// TIA Portal V16 export
// export: Created 2021-11-12T13:32:31.7441446Z, ExportSetting WithDefaults, DisplayName Totally Integrated Automation Portal, DisplayVersion V16 Update 3, DisplayName TIA Portal Version Control Interface, DisplayVersion V16 Update 2, DisplayName TIA Portal Openness, DisplayVersion V16 Update 3, DisplayName SINAMICS Startdrive Advanced, DisplayVersion V16 Update 5, DisplayName SINAMICS Startdrive G130, G150, S120, S150, SINAMICS MV, S210, DisplayVersion V16 Update 5, DisplayName SINAMICS Startdrive G110M, G120, G120C, G120D, G120P, G115D, DisplayVersion V16 Update 5, DisplayName STEP 7 Professional, DisplayVersion V16 Update 3, DisplayName STEP 7 Safety, DisplayVersion V16, DisplayName WinCC UA Professional, DisplayVersion V16 Update 3
FUNCTION_BLOCK "IM_100+UH13-KF10"   // FB62, LAD
TITLE = Inputs reading
{ S7_Optimized_Access := 'TRUE' }
VERSION : 0.1
// MICE Wood interface block
// stored: AutoNumber true, IsIECCheckEnabled false, IsRetainMemResEnabled false, MemoryReserve 100, SetENOAutomatically false, UDAEnableTagReadback false
   VAR
      KF11_Ix0 { S7_SetPoint := 'True'} : "STD_CH_DI";
      KF11_Ix1 { S7_SetPoint := 'True'} : "STD_CH_DI";
      KF11_Ix2 { S7_SetPoint := 'True'} : "STD_CH_DI";
      KF11_Ix3 { S7_SetPoint := 'True'} : "STD_CH_DI";
      KF11_Ix4 { S7_SetPoint := 'True'} : "STD_CH_DI";
      KF11_Ix5 { S7_SetPoint := 'True'} : "STD_CH_DI";
      KF11_Ix6 { S7_SetPoint := 'True'} : "STD_CH_DI";
      KF11_Ix7 { S7_SetPoint := 'True'} : "STD_CH_DI";
      KF11_Ix8 { S7_SetPoint := 'True'} : "STD_CH_DI";
      KF11_Ix9 { S7_SetPoint := 'True'} : "STD_CH_DI";
      KF11_Ix10 { S7_SetPoint := 'True'} : "STD_CH_DI";
      KF11_Ix11 { S7_SetPoint := 'True'} : "STD_CH_DI";
      KF11_Ix12 { S7_SetPoint := 'True'} : "STD_CH_DI";
      KF11_Ix13 { S7_SetPoint := 'True'} : "STD_CH_DI";
      KF11_Ix14 { S7_SetPoint := 'True'} : "STD_CH_DI";
      KF11_Ix15 { S7_SetPoint := 'True'} : "STD_CH_DI";
      KF12_Ix0 { S7_SetPoint := 'True'} : "STD_CH_DI";
      KF12_Ix1 { S7_SetPoint := 'True'} : "STD_CH_DI";
      KF12_Ix2 { S7_SetPoint := 'True'} : "STD_CH_DI";
      KF12_Ix3 { S7_SetPoint := 'True'} : "STD_CH_DI";
      KF12_Ix4 { S7_SetPoint := 'True'} : "STD_CH_DI";
      KF12_Ix5 { S7_SetPoint := 'True'} : "STD_CH_DI";
      KF12_Ix6 { S7_SetPoint := 'True'} : "STD_CH_DI";
      KF12_Ix7 { S7_SetPoint := 'True'} : "STD_CH_DI";
      KF12_Ix8 { S7_SetPoint := 'True'} : "STD_CH_DI";
      KF12_Ix9 { S7_SetPoint := 'True'} : "STD_CH_DI";
      KF12_Ix10 { S7_SetPoint := 'True'} : "STD_CH_DI";
      KF12_Ix11 { S7_SetPoint := 'True'} : "STD_CH_DI";
      KF12_Ix12 { S7_SetPoint := 'True'} : "STD_CH_DI";
      KF12_Ix13 { S7_SetPoint := 'True'} : "STD_CH_DI";
      KF12_Ix14 { S7_SetPoint := 'True'} : "STD_CH_DI";
      KF12_Ix15 { S7_SetPoint := 'True'} : "STD_CH_DI";
   END_VAR
   VAR_TEMP   // added for the SCL form of the ladder/FBD networks
      _w1 : Bool;
      _w2 : Bool;
      _w3 : Bool;
      _w4 : Bool;
      _w5 : Bool;
      _w6 : Bool;
      _w7 : Bool;
   END_VAR
BEGIN

REGION Network 1: Module position -KF11
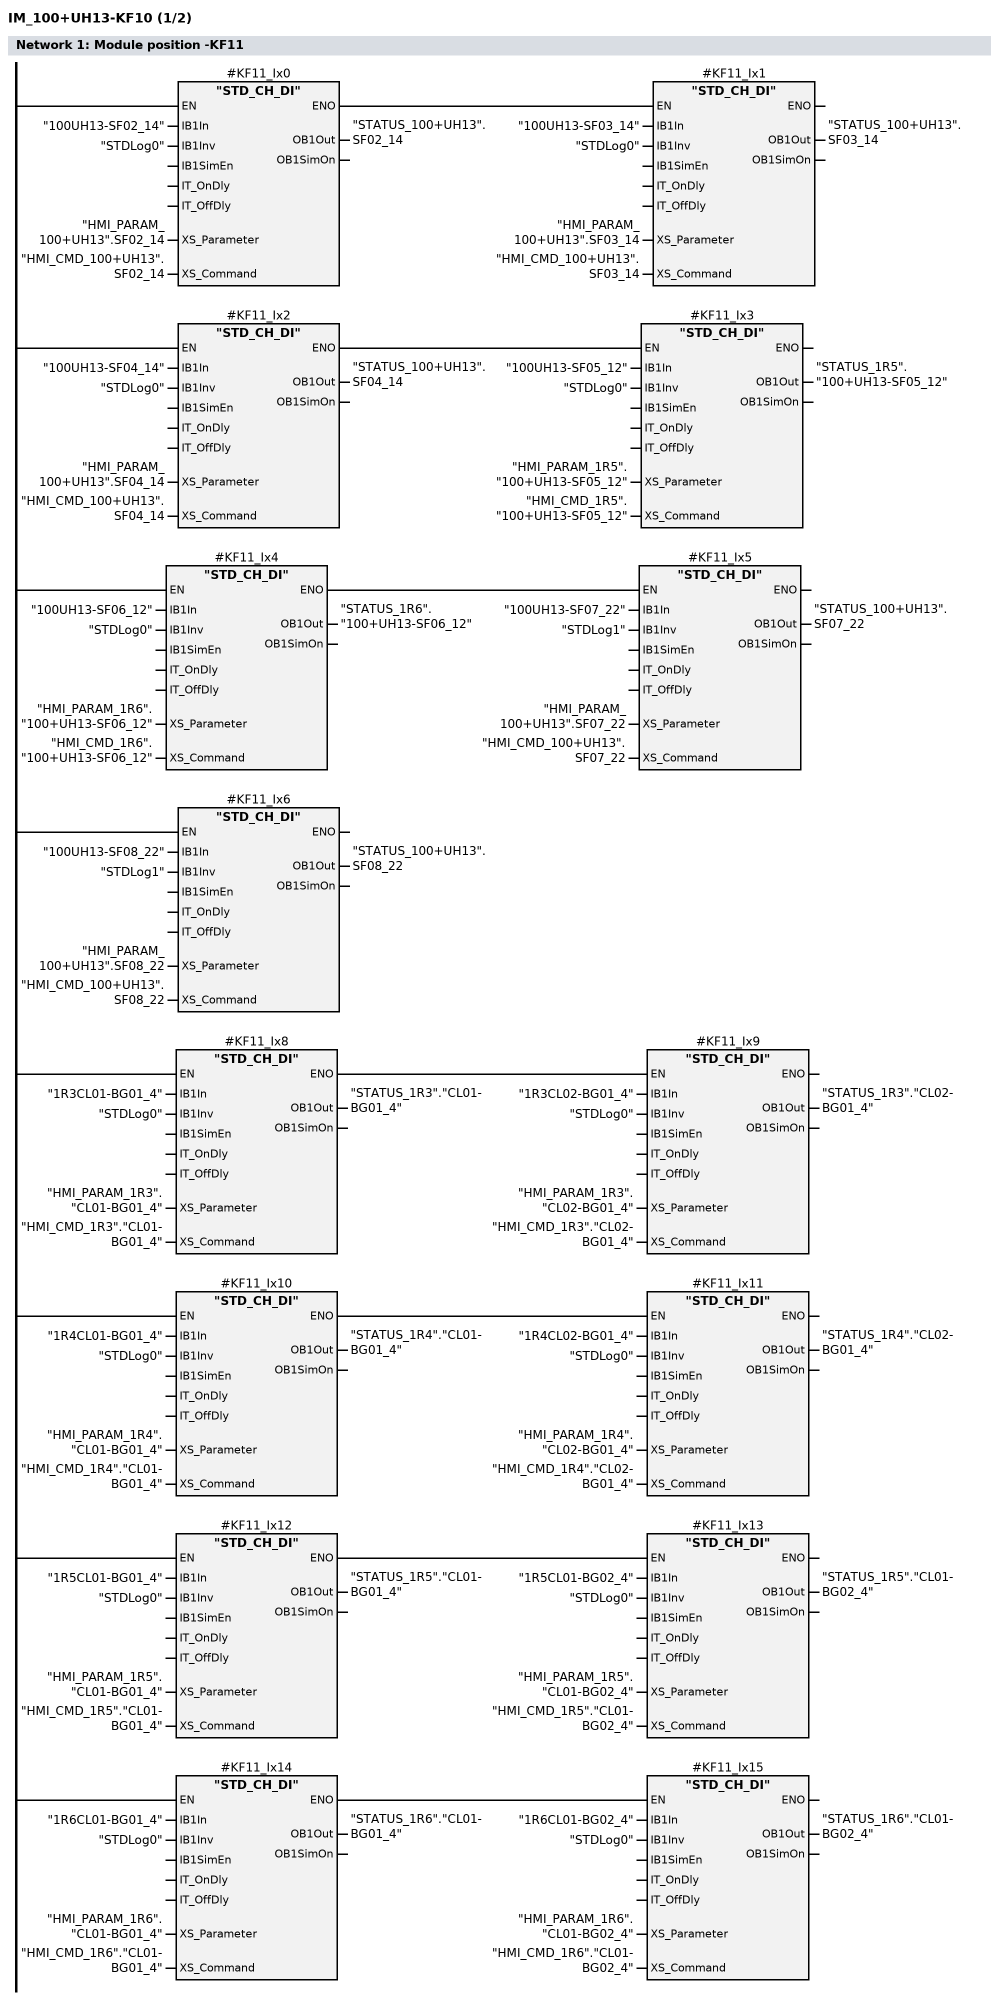
   RUNG wire#powerrail
      #KF11_Ix0(IB1In := "100UH13-SF02_14", IB1Inv := "STDLog0", IB1SimEn :=, IT_OnDly :=, IT_OffDly :=, XS_Parameter := "HMI_PARAM_100+UH13".SF02_14, XS_Command := "HMI_CMD_100+UH13".SF02_14, OB1Out => "STATUS_100+UH13".SF02_14, OB1SimOn =>)
      #KF11_Ix1(IB1In := "100UH13-SF03_14", IB1Inv := "STDLog0", IB1SimEn :=, IT_OnDly :=, IT_OffDly :=, XS_Parameter := "HMI_PARAM_100+UH13".SF03_14, XS_Command := "HMI_CMD_100+UH13".SF03_14, OB1Out => "STATUS_100+UH13".SF03_14, OB1SimOn =>)
   END_RUNG
   RUNG wire#powerrail
      #KF11_Ix2(IB1In := "100UH13-SF04_14", IB1Inv := "STDLog0", IB1SimEn :=, IT_OnDly :=, IT_OffDly :=, XS_Parameter := "HMI_PARAM_100+UH13".SF04_14, XS_Command := "HMI_CMD_100+UH13".SF04_14, OB1Out => "STATUS_100+UH13".SF04_14, OB1SimOn =>)
      #KF11_Ix3(IB1In := "100UH13-SF05_12", IB1Inv := "STDLog0", IB1SimEn :=, IT_OnDly :=, IT_OffDly :=, XS_Parameter := "HMI_PARAM_1R5"."100+UH13-SF05_12", XS_Command := "HMI_CMD_1R5"."100+UH13-SF05_12", OB1Out => "STATUS_1R5"."100+UH13-SF05_12", OB1SimOn =>)
   END_RUNG
   RUNG wire#powerrail
      #KF11_Ix4(IB1In := "100UH13-SF06_12", IB1Inv := "STDLog0", IB1SimEn :=, IT_OnDly :=, IT_OffDly :=, XS_Parameter := "HMI_PARAM_1R6"."100+UH13-SF06_12", XS_Command := "HMI_CMD_1R6"."100+UH13-SF06_12", OB1Out => "STATUS_1R6"."100+UH13-SF06_12", OB1SimOn =>)
      #KF11_Ix5(IB1In := "100UH13-SF07_22", IB1Inv := "STDLog1", IB1SimEn :=, IT_OnDly :=, IT_OffDly :=, XS_Parameter := "HMI_PARAM_100+UH13".SF07_22, XS_Command := "HMI_CMD_100+UH13".SF07_22, OB1Out => "STATUS_100+UH13".SF07_22, OB1SimOn =>)
   END_RUNG
   RUNG wire#powerrail
      #KF11_Ix6(IB1In := "100UH13-SF08_22", IB1Inv := "STDLog1", IB1SimEn :=, IT_OnDly :=, IT_OffDly :=, XS_Parameter := "HMI_PARAM_100+UH13".SF08_22, XS_Command := "HMI_CMD_100+UH13".SF08_22, OB1Out => "STATUS_100+UH13".SF08_22, OB1SimOn =>)
   END_RUNG
   RUNG wire#powerrail
      #KF11_Ix8(IB1In := "1R3CL01-BG01_4", IB1Inv := "STDLog0", IB1SimEn :=, IT_OnDly :=, IT_OffDly :=, XS_Parameter := "HMI_PARAM_1R3"."CL01-BG01_4", XS_Command := "HMI_CMD_1R3"."CL01-BG01_4", OB1Out => "STATUS_1R3"."CL01-BG01_4", OB1SimOn =>)
      #KF11_Ix9(IB1In := "1R3CL02-BG01_4", IB1Inv := "STDLog0", IB1SimEn :=, IT_OnDly :=, IT_OffDly :=, XS_Parameter := "HMI_PARAM_1R3"."CL02-BG01_4", XS_Command := "HMI_CMD_1R3"."CL02-BG01_4", OB1Out => "STATUS_1R3"."CL02-BG01_4", OB1SimOn =>)
   END_RUNG
   RUNG wire#powerrail
      #KF11_Ix10(IB1In := "1R4CL01-BG01_4", IB1Inv := "STDLog0", IB1SimEn :=, IT_OnDly :=, IT_OffDly :=, XS_Parameter := "HMI_PARAM_1R4"."CL01-BG01_4", XS_Command := "HMI_CMD_1R4"."CL01-BG01_4", OB1Out => "STATUS_1R4"."CL01-BG01_4", OB1SimOn =>)
      #KF11_Ix11(IB1In := "1R4CL02-BG01_4", IB1Inv := "STDLog0", IB1SimEn :=, IT_OnDly :=, IT_OffDly :=, XS_Parameter := "HMI_PARAM_1R4"."CL02-BG01_4", XS_Command := "HMI_CMD_1R4"."CL02-BG01_4", OB1Out => "STATUS_1R4"."CL02-BG01_4", OB1SimOn =>)
   END_RUNG
   RUNG wire#powerrail
      #KF11_Ix12(IB1In := "1R5CL01-BG01_4", IB1Inv := "STDLog0", IB1SimEn :=, IT_OnDly :=, IT_OffDly :=, XS_Parameter := "HMI_PARAM_1R5"."CL01-BG01_4", XS_Command := "HMI_CMD_1R5"."CL01-BG01_4", OB1Out => "STATUS_1R5"."CL01-BG01_4", OB1SimOn =>)
      #KF11_Ix13(IB1In := "1R5CL01-BG02_4", IB1Inv := "STDLog0", IB1SimEn :=, IT_OnDly :=, IT_OffDly :=, XS_Parameter := "HMI_PARAM_1R5"."CL01-BG02_4", XS_Command := "HMI_CMD_1R5"."CL01-BG02_4", OB1Out => "STATUS_1R5"."CL01-BG02_4", OB1SimOn =>)
   END_RUNG
   RUNG wire#powerrail
      #KF11_Ix14(IB1In := "1R6CL01-BG01_4", IB1Inv := "STDLog0", IB1SimEn :=, IT_OnDly :=, IT_OffDly :=, XS_Parameter := "HMI_PARAM_1R6"."CL01-BG01_4", XS_Command := "HMI_CMD_1R6"."CL01-BG01_4", OB1Out => "STATUS_1R6"."CL01-BG01_4", OB1SimOn =>)
      #KF11_Ix15(IB1In := "1R6CL01-BG02_4", IB1Inv := "STDLog0", IB1SimEn :=, IT_OnDly :=, IT_OffDly :=, XS_Parameter := "HMI_PARAM_1R6"."CL01-BG02_4", XS_Command := "HMI_CMD_1R6"."CL01-BG02_4", OB1Out => "STATUS_1R6"."CL01-BG02_4", OB1SimOn =>)
   END_RUNG
   // the same network as SCL:
   #KF11_Ix0(IB1In := "100UH13-SF02_14",   // "STD_CH_DI"
             IB1Inv := "STDLog0",
             XS_Parameter := "HMI_PARAM_100+UH13".SF02_14,
             XS_Command := "HMI_CMD_100+UH13".SF02_14,
             OB1Out => "STATUS_100+UH13".SF02_14,
             ENO => #_w1);
   IF #_w1 THEN
       #KF11_Ix1(IB1In := "100UH13-SF03_14",   // "STD_CH_DI"
                 IB1Inv := "STDLog0",
                 XS_Parameter := "HMI_PARAM_100+UH13".SF03_14,
                 XS_Command := "HMI_CMD_100+UH13".SF03_14,
                 OB1Out => "STATUS_100+UH13".SF03_14);
   END_IF;
   #KF11_Ix2(IB1In := "100UH13-SF04_14",   // "STD_CH_DI"
             IB1Inv := "STDLog0",
             XS_Parameter := "HMI_PARAM_100+UH13".SF04_14,
             XS_Command := "HMI_CMD_100+UH13".SF04_14,
             OB1Out => "STATUS_100+UH13".SF04_14,
             ENO => #_w2);
   IF #_w2 THEN
       #KF11_Ix3(IB1In := "100UH13-SF05_12",   // "STD_CH_DI"
                 IB1Inv := "STDLog0",
                 XS_Parameter := "HMI_PARAM_1R5"."100+UH13-SF05_12",
                 XS_Command := "HMI_CMD_1R5"."100+UH13-SF05_12",
                 OB1Out => "STATUS_1R5"."100+UH13-SF05_12");
   END_IF;
   #KF11_Ix4(IB1In := "100UH13-SF06_12",   // "STD_CH_DI"
             IB1Inv := "STDLog0",
             XS_Parameter := "HMI_PARAM_1R6"."100+UH13-SF06_12",
             XS_Command := "HMI_CMD_1R6"."100+UH13-SF06_12",
             OB1Out => "STATUS_1R6"."100+UH13-SF06_12",
             ENO => #_w3);
   IF #_w3 THEN
       #KF11_Ix5(IB1In := "100UH13-SF07_22",   // "STD_CH_DI"
                 IB1Inv := "STDLog1",
                 XS_Parameter := "HMI_PARAM_100+UH13".SF07_22,
                 XS_Command := "HMI_CMD_100+UH13".SF07_22,
                 OB1Out => "STATUS_100+UH13".SF07_22);
   END_IF;
   #KF11_Ix6(IB1In := "100UH13-SF08_22",   // "STD_CH_DI"
             IB1Inv := "STDLog1",
             XS_Parameter := "HMI_PARAM_100+UH13".SF08_22,
             XS_Command := "HMI_CMD_100+UH13".SF08_22,
             OB1Out => "STATUS_100+UH13".SF08_22);
   #KF11_Ix8(IB1In := "1R3CL01-BG01_4",   // "STD_CH_DI"
             IB1Inv := "STDLog0",
             XS_Parameter := "HMI_PARAM_1R3"."CL01-BG01_4",
             XS_Command := "HMI_CMD_1R3"."CL01-BG01_4",
             OB1Out => "STATUS_1R3"."CL01-BG01_4",
             ENO => #_w4);
   IF #_w4 THEN
       #KF11_Ix9(IB1In := "1R3CL02-BG01_4",   // "STD_CH_DI"
                 IB1Inv := "STDLog0",
                 XS_Parameter := "HMI_PARAM_1R3"."CL02-BG01_4",
                 XS_Command := "HMI_CMD_1R3"."CL02-BG01_4",
                 OB1Out => "STATUS_1R3"."CL02-BG01_4");
   END_IF;
   #KF11_Ix10(IB1In := "1R4CL01-BG01_4",   // "STD_CH_DI"
              IB1Inv := "STDLog0",
              XS_Parameter := "HMI_PARAM_1R4"."CL01-BG01_4",
              XS_Command := "HMI_CMD_1R4"."CL01-BG01_4",
              OB1Out => "STATUS_1R4"."CL01-BG01_4",
              ENO => #_w5);
   IF #_w5 THEN
       #KF11_Ix11(IB1In := "1R4CL02-BG01_4",   // "STD_CH_DI"
                  IB1Inv := "STDLog0",
                  XS_Parameter := "HMI_PARAM_1R4"."CL02-BG01_4",
                  XS_Command := "HMI_CMD_1R4"."CL02-BG01_4",
                  OB1Out => "STATUS_1R4"."CL02-BG01_4");
   END_IF;
   #KF11_Ix12(IB1In := "1R5CL01-BG01_4",   // "STD_CH_DI"
              IB1Inv := "STDLog0",
              XS_Parameter := "HMI_PARAM_1R5"."CL01-BG01_4",
              XS_Command := "HMI_CMD_1R5"."CL01-BG01_4",
              OB1Out => "STATUS_1R5"."CL01-BG01_4",
              ENO => #_w6);
   IF #_w6 THEN
       #KF11_Ix13(IB1In := "1R5CL01-BG02_4",   // "STD_CH_DI"
                  IB1Inv := "STDLog0",
                  XS_Parameter := "HMI_PARAM_1R5"."CL01-BG02_4",
                  XS_Command := "HMI_CMD_1R5"."CL01-BG02_4",
                  OB1Out => "STATUS_1R5"."CL01-BG02_4");
   END_IF;
   #KF11_Ix14(IB1In := "1R6CL01-BG01_4",   // "STD_CH_DI"
              IB1Inv := "STDLog0",
              XS_Parameter := "HMI_PARAM_1R6"."CL01-BG01_4",
              XS_Command := "HMI_CMD_1R6"."CL01-BG01_4",
              OB1Out => "STATUS_1R6"."CL01-BG01_4",
              ENO => #_w7);
   IF #_w7 THEN
       #KF11_Ix15(IB1In := "1R6CL01-BG02_4",   // "STD_CH_DI"
                  IB1Inv := "STDLog0",
                  XS_Parameter := "HMI_PARAM_1R6"."CL01-BG02_4",
                  XS_Command := "HMI_CMD_1R6"."CL01-BG02_4",
                  OB1Out => "STATUS_1R6"."CL01-BG02_4");
   END_IF;
END_REGION

REGION Network 2: Module position -KF12
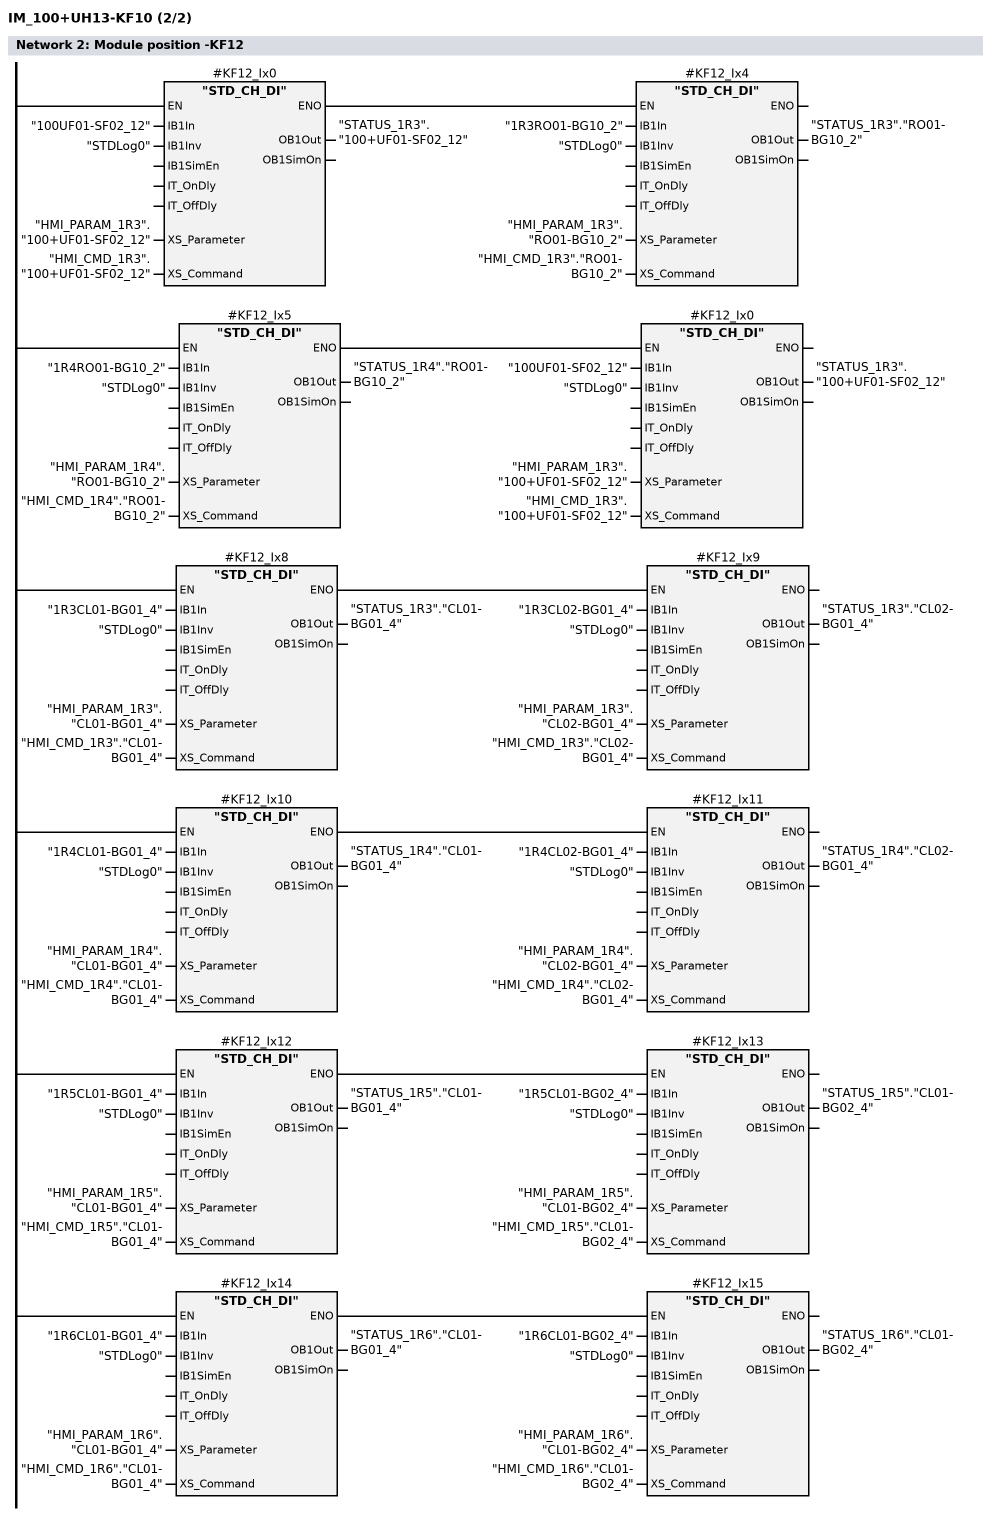
   RUNG wire#powerrail
      #KF12_Ix0(IB1In := "100UF01-SF02_12", IB1Inv := "STDLog0", IB1SimEn :=, IT_OnDly :=, IT_OffDly :=, XS_Parameter := "HMI_PARAM_1R3"."100+UF01-SF02_12", XS_Command := "HMI_CMD_1R3"."100+UF01-SF02_12", OB1Out => "STATUS_1R3"."100+UF01-SF02_12", OB1SimOn =>)
      #KF12_Ix4(IB1In := "1R3RO01-BG10_2", IB1Inv := "STDLog0", IB1SimEn :=, IT_OnDly :=, IT_OffDly :=, XS_Parameter := "HMI_PARAM_1R3"."RO01-BG10_2", XS_Command := "HMI_CMD_1R3"."RO01-BG10_2", OB1Out => "STATUS_1R3"."RO01-BG10_2", OB1SimOn =>)
   END_RUNG
   RUNG wire#powerrail
      #KF12_Ix5(IB1In := "1R4RO01-BG10_2", IB1Inv := "STDLog0", IB1SimEn :=, IT_OnDly :=, IT_OffDly :=, XS_Parameter := "HMI_PARAM_1R4"."RO01-BG10_2", XS_Command := "HMI_CMD_1R4"."RO01-BG10_2", OB1Out => "STATUS_1R4"."RO01-BG10_2", OB1SimOn =>)
      #KF12_Ix0(IB1In := "100UF01-SF02_12", IB1Inv := "STDLog0", IB1SimEn :=, IT_OnDly :=, IT_OffDly :=, XS_Parameter := "HMI_PARAM_1R3"."100+UF01-SF02_12", XS_Command := "HMI_CMD_1R3"."100+UF01-SF02_12", OB1Out => "STATUS_1R3"."100+UF01-SF02_12", OB1SimOn =>)
   END_RUNG
   RUNG wire#powerrail
      #KF12_Ix8(IB1In := "1R3CL01-BG01_4", IB1Inv := "STDLog0", IB1SimEn :=, IT_OnDly :=, IT_OffDly :=, XS_Parameter := "HMI_PARAM_1R3"."CL01-BG01_4", XS_Command := "HMI_CMD_1R3"."CL01-BG01_4", OB1Out => "STATUS_1R3"."CL01-BG01_4", OB1SimOn =>)
      #KF12_Ix9(IB1In := "1R3CL02-BG01_4", IB1Inv := "STDLog0", IB1SimEn :=, IT_OnDly :=, IT_OffDly :=, XS_Parameter := "HMI_PARAM_1R3"."CL02-BG01_4", XS_Command := "HMI_CMD_1R3"."CL02-BG01_4", OB1Out => "STATUS_1R3"."CL02-BG01_4", OB1SimOn =>)
   END_RUNG
   RUNG wire#powerrail
      #KF12_Ix10(IB1In := "1R4CL01-BG01_4", IB1Inv := "STDLog0", IB1SimEn :=, IT_OnDly :=, IT_OffDly :=, XS_Parameter := "HMI_PARAM_1R4"."CL01-BG01_4", XS_Command := "HMI_CMD_1R4"."CL01-BG01_4", OB1Out => "STATUS_1R4"."CL01-BG01_4", OB1SimOn =>)
      #KF12_Ix11(IB1In := "1R4CL02-BG01_4", IB1Inv := "STDLog0", IB1SimEn :=, IT_OnDly :=, IT_OffDly :=, XS_Parameter := "HMI_PARAM_1R4"."CL02-BG01_4", XS_Command := "HMI_CMD_1R4"."CL02-BG01_4", OB1Out => "STATUS_1R4"."CL02-BG01_4", OB1SimOn =>)
   END_RUNG
   RUNG wire#powerrail
      #KF12_Ix12(IB1In := "1R5CL01-BG01_4", IB1Inv := "STDLog0", IB1SimEn :=, IT_OnDly :=, IT_OffDly :=, XS_Parameter := "HMI_PARAM_1R5"."CL01-BG01_4", XS_Command := "HMI_CMD_1R5"."CL01-BG01_4", OB1Out => "STATUS_1R5"."CL01-BG01_4", OB1SimOn =>)
      #KF12_Ix13(IB1In := "1R5CL01-BG02_4", IB1Inv := "STDLog0", IB1SimEn :=, IT_OnDly :=, IT_OffDly :=, XS_Parameter := "HMI_PARAM_1R5"."CL01-BG02_4", XS_Command := "HMI_CMD_1R5"."CL01-BG02_4", OB1Out => "STATUS_1R5"."CL01-BG02_4", OB1SimOn =>)
   END_RUNG
   RUNG wire#powerrail
      #KF12_Ix14(IB1In := "1R6CL01-BG01_4", IB1Inv := "STDLog0", IB1SimEn :=, IT_OnDly :=, IT_OffDly :=, XS_Parameter := "HMI_PARAM_1R6"."CL01-BG01_4", XS_Command := "HMI_CMD_1R6"."CL01-BG01_4", OB1Out => "STATUS_1R6"."CL01-BG01_4", OB1SimOn =>)
      #KF12_Ix15(IB1In := "1R6CL01-BG02_4", IB1Inv := "STDLog0", IB1SimEn :=, IT_OnDly :=, IT_OffDly :=, XS_Parameter := "HMI_PARAM_1R6"."CL01-BG02_4", XS_Command := "HMI_CMD_1R6"."CL01-BG02_4", OB1Out => "STATUS_1R6"."CL01-BG02_4", OB1SimOn =>)
   END_RUNG
   // the same network as SCL:
   #KF12_Ix0(IB1In := "100UF01-SF02_12",   // "STD_CH_DI"
             IB1Inv := "STDLog0",
             XS_Parameter := "HMI_PARAM_1R3"."100+UF01-SF02_12",
             XS_Command := "HMI_CMD_1R3"."100+UF01-SF02_12",
             OB1Out => "STATUS_1R3"."100+UF01-SF02_12",
             ENO => #_w1);
   IF #_w1 THEN
       #KF12_Ix4(IB1In := "1R3RO01-BG10_2",   // "STD_CH_DI"
                 IB1Inv := "STDLog0",
                 XS_Parameter := "HMI_PARAM_1R3"."RO01-BG10_2",
                 XS_Command := "HMI_CMD_1R3"."RO01-BG10_2",
                 OB1Out => "STATUS_1R3"."RO01-BG10_2");
   END_IF;
   #KF12_Ix5(IB1In := "1R4RO01-BG10_2",   // "STD_CH_DI"
             IB1Inv := "STDLog0",
             XS_Parameter := "HMI_PARAM_1R4"."RO01-BG10_2",
             XS_Command := "HMI_CMD_1R4"."RO01-BG10_2",
             OB1Out => "STATUS_1R4"."RO01-BG10_2",
             ENO => #_w2);
   IF #_w2 THEN
       #KF12_Ix0(IB1In := "100UF01-SF02_12",   // "STD_CH_DI"
                 IB1Inv := "STDLog0",
                 XS_Parameter := "HMI_PARAM_1R3"."100+UF01-SF02_12",
                 XS_Command := "HMI_CMD_1R3"."100+UF01-SF02_12",
                 OB1Out => "STATUS_1R3"."100+UF01-SF02_12");
   END_IF;
   #KF12_Ix8(IB1In := "1R3CL01-BG01_4",   // "STD_CH_DI"
             IB1Inv := "STDLog0",
             XS_Parameter := "HMI_PARAM_1R3"."CL01-BG01_4",
             XS_Command := "HMI_CMD_1R3"."CL01-BG01_4",
             OB1Out => "STATUS_1R3"."CL01-BG01_4",
             ENO => #_w3);
   IF #_w3 THEN
       #KF12_Ix9(IB1In := "1R3CL02-BG01_4",   // "STD_CH_DI"
                 IB1Inv := "STDLog0",
                 XS_Parameter := "HMI_PARAM_1R3"."CL02-BG01_4",
                 XS_Command := "HMI_CMD_1R3"."CL02-BG01_4",
                 OB1Out => "STATUS_1R3"."CL02-BG01_4");
   END_IF;
   #KF12_Ix10(IB1In := "1R4CL01-BG01_4",   // "STD_CH_DI"
              IB1Inv := "STDLog0",
              XS_Parameter := "HMI_PARAM_1R4"."CL01-BG01_4",
              XS_Command := "HMI_CMD_1R4"."CL01-BG01_4",
              OB1Out => "STATUS_1R4"."CL01-BG01_4",
              ENO => #_w4);
   IF #_w4 THEN
       #KF12_Ix11(IB1In := "1R4CL02-BG01_4",   // "STD_CH_DI"
                  IB1Inv := "STDLog0",
                  XS_Parameter := "HMI_PARAM_1R4"."CL02-BG01_4",
                  XS_Command := "HMI_CMD_1R4"."CL02-BG01_4",
                  OB1Out => "STATUS_1R4"."CL02-BG01_4");
   END_IF;
   #KF12_Ix12(IB1In := "1R5CL01-BG01_4",   // "STD_CH_DI"
              IB1Inv := "STDLog0",
              XS_Parameter := "HMI_PARAM_1R5"."CL01-BG01_4",
              XS_Command := "HMI_CMD_1R5"."CL01-BG01_4",
              OB1Out => "STATUS_1R5"."CL01-BG01_4",
              ENO => #_w5);
   IF #_w5 THEN
       #KF12_Ix13(IB1In := "1R5CL01-BG02_4",   // "STD_CH_DI"
                  IB1Inv := "STDLog0",
                  XS_Parameter := "HMI_PARAM_1R5"."CL01-BG02_4",
                  XS_Command := "HMI_CMD_1R5"."CL01-BG02_4",
                  OB1Out => "STATUS_1R5"."CL01-BG02_4");
   END_IF;
   #KF12_Ix14(IB1In := "1R6CL01-BG01_4",   // "STD_CH_DI"
              IB1Inv := "STDLog0",
              XS_Parameter := "HMI_PARAM_1R6"."CL01-BG01_4",
              XS_Command := "HMI_CMD_1R6"."CL01-BG01_4",
              OB1Out => "STATUS_1R6"."CL01-BG01_4",
              ENO => #_w6);
   IF #_w6 THEN
       #KF12_Ix15(IB1In := "1R6CL01-BG02_4",   // "STD_CH_DI"
                  IB1Inv := "STDLog0",
                  XS_Parameter := "HMI_PARAM_1R6"."CL01-BG02_4",
                  XS_Command := "HMI_CMD_1R6"."CL01-BG02_4",
                  OB1Out => "STATUS_1R6"."CL01-BG02_4");
   END_IF;
END_REGION
END_FUNCTION_BLOCK
